{attribute 'reflection'}
FUNCTION_BLOCK PUBLIC FB_DevDoublePWM EXTENDS FB_DevBase // PWM control for 2 outputs that cannot be switchid on simultaniously
VAR_INPUT
	bCmdPWMOn			: BOOL := FALSE ; // PWM controller on 
END_VAR
VAR_OUTPUT
END_VAR
VAR
	bCmdChanelAOn		: BOOL := FALSE ; // command switch chanel A on permanently
	bCmdChanelBOn		: BOOL := FALSE ; // Commandswitch chanel B on permanently 
	bCmdOverrulePWM		: BOOL := FALSE ; // Command to overrule PWM
	bCmdHold			: BOOL := false ; // Command hold PWM on signals (collision avoidance)

	tPeriodLength		: TIME  ; // desired PWM cycle time length [ms] 
	tDutyCycle 			: TIME	; // percentage of power [%]
	tIdleTime			: TIME	; // Time both outputs are idle during PWM
	
	tonOutputA 			: TON ; // Timer on PWM output A
	tonOutputB 			: TON ; // Timer on PWM output B
	tonIdle				: TON ; // Timer On PWM Idle time (both outputs off)

	tofOutputA 			: TOF ; // Timer off PWM output A Off (For overlap prevention)
	tofOutputB 			: TOF ; // Timer off PWM output B Off ( for overlap prevention)

	stParPeriodLength	: Udt_Parameter := (fValue := 2000); // desired PWM cycle time length [ms] Parameter
	stParDutyCycle 		: Udt_Parameter	:= ( fValue := 0); // percentage of power [%] Parameter
	stParSwitchOverTime	: Udt_Parameter	; // Time between switching A off and B on (and vice versa) Parameter
	stMaxTimeOn			: Udt_Parameter := (fValue := 1000);// Maximum time a heater can be on without burning through
	
	qbOutputMain AT %Q* 	: BOOL 	; // physical output to main relais
	qbOutputA	 AT %Q* 	: BOOL 	; // physical output to output A
	qbOutputB	 AT %Q* 	: BOOL 	; // physical output to output B
	
	nPWMStep	: INT ; // PWM stepper

	tonBurnTimeA	: TON ; // burn timer for coil A
	tonBurnTimeB	: TON ; // burn timer for coil B 
END_VAR

// set device type
IF eDevType = E_Devices.Undefined THEN 
	eDevType := E_Devices.DoublePWMController ;
END_IF

// Call base function
SUPER^();


// ===== hold all actions if not initialized ======
IF NOT bInitOk THEN
	RETURN;
END_IF 

// call Functions 
CalcCycleTimes();
IF tDutyCycle > T#0S AND tPeriodLength > T#0S THEN // switch PWM controller up when cycle timer is null
	ExecPWMCycle(); // 
END_IF 

ExecSetOutputs();

METHOD INTERNAL CalcCycleTimes : BOOL // calculate cycle timers
VAR_INPUT
END_VAR
VAR 
END_VAR
// Calculate Cycle timers
tPeriodLength	:= LREAL_TO_TIME( stParPeriodLength.fValue );
tDutyCycle		:= LREAL_TO_TIME(stParPeriodLength.fValue * (stParDutyCycle.fValue / 100));
tIdleTime		:= LREAL_TO_TIME(stParPeriodLength.fValue) - (tDutyCycle * 2) ;

tofOutputA.PT := LREAL_TO_TIME(stParSwitchOverTime.fValue);
tofOutputB.PT := LREAL_TO_TIME(stParSwitchOverTime.fValue);
END_METHOD

METHOD PUBLIC CmdHold : BOOL
VAR_INPUT
END_VAR
bCmdHold := TRUE ;

CmdHold := NOT qbOutputMain ;
END_METHOD

METHOD PUBLIC CmdOutputAOn : BOOL // Turn on chanel A permanently 
VAR_INPUT
END_VAR
bCmdOverrulePWM S= TRUE ;
bCmdChanelAOn S= TRUE ;

CmdOutputAOn := qbOutputA AND qbOutputMain ;
END_METHOD

METHOD PUBLIC CmdOutputBOn : BOOL
VAR_INPUT
END_VAR
bCmdOverrulePWM S= TRUE ;
bCmdChanelBOn S= TRUE ;

CmdOutputBOn := qbOutputB AND qbOutputMain ;
END_METHOD

METHOD PUBLIC CmdSafeStop : BOOL
VAR_INPUT
END_VAR
bCmdOverrulePWM S= TRUE ;
bCmdChanelAOn 		:= FALSE ;
bCmdChanelBOn		:= FALSE ;
qbOutputMain 		:= FALSE ;

bIsSafe := NOT (qbOutputA OR qbOutputB OR qbOutputMain);
END_METHOD

METHOD INTERNAL ExecPWMCycle : BOOL
VAR_INPUT
END_VAR
IF bCmdPWMOn THEN 
	IF bCmdOverrulePWM OR bCmdHold THEN 
		IF bCmdChanelAOn THEN 
			nPWMStep := 1 ;
		ELSE 
			nPWMStep := 0 ;
		END_IF
		bCmdOverrulePWM := FALSE ;
		RETURN;
	END_IF
ELSE 
	RETURN;
END_IF

// PWM stepper 
CASE nPWMStep OF 
	0: // Switch on chanel A
		bCmdChanelAOn := TRUE ;
		IF tonOutputA.Q THEN
			nPWMStep := 1 ;
		END_IF
	1: // Switch on chanel B
		bCmdChanelBOn := TRUE;
		IF tonOutputB.Q THEN
			nPWMStep := 2 ;
		END_IF
	2: // Idle Time 
		IF tonIdle.Q THEN 
			nPWMStep := 0;
		END_IF
	ELSE
		;
END_CASE

// call timers 
tonOutputA	(IN := bCmdChanelAOn, PT := tDutyCycle);
tonOutputB	(IN := bCmdChanelBOn, PT := tDutyCycle);
tonIdle 	(IN := nPWMStep = 2	, PT := tIdleTime);
END_METHOD

METHOD PRIVATE ExecSetOutputs : BOOL
VAR_INPUT
END_VAR

// Set main output
qbOutputMain := (bEnable OR bManual) AND NOT bCmdHold ;

// Set outputs
qbOutputA := bCmdChanelAOn AND NOT tofOutputB.Q AND NOT tonBurnTimeA.Q;
qbOutputB := bCmdChanelBOn AND NOT tofOutputA.Q AND NOT tonBurnTimeB.Q;

// Call timers for overlap prevention
tofOutputA(IN := qbOutputA);
tofOutputB(IN := qbOutputB);

// reset commands
bCmdChanelAOn := FALSE ;
bCmdChanelBOn := FALSE ;

tonBurnTimeA ( IN := bCmdChanelAOn, PT := LREAL_TO_TIME( stMaxTimeOn.fValue));
tonBurnTimeB ( IN := bCmdChanelBOn, PT := LREAL_TO_TIME( stMaxTimeOn.fValue));

IF tonBurnTimeA.Q THEN 
	stFault.Active 			:= TRUE ;
	stFault.Description 	:= 'Heater A burn timeout';
	stFault.FaultType		:= E_FaultTypes.CF;
	qbOutputA 				:= FALSE ;
ELSIF tonBurnTimeB.Q THEN 
	stFault.Active 			:= TRUE ;
	stFault.Description 	:= 'Heater B burn timeout';
	stFault.FaultType		:= E_FaultTypes.CF;
	qbOutputB 				:= FALSE ;
END_IF

bCmdHold := FALSE ;
END_METHOD

METHOD PUBLIC Init : BOOL
VAR_INPUT
	// Message location data
	nId			: UINT ; // Identification number of object
	nParentId	: UDINT ; // Id of higher level If aplicable (0 = no parent)
END_VAR
// ====== Set init to true =====
	bInitOk	:= TRUE ; 

// ====== Calculate device id =====
	bInitOk :=	ExecIdentifyDevice(nId,nParentId, E_ComponentTypes.Heaters) AND bInitOk;

// ======= Reset Error bit ======
	bErrorActive 	:= FALSE;
	bBusy			:= FALSE;
	
// ===== configure parameters =====
	stParPeriodLength.fMinimum 		:= 0 		;
	stParPeriodLength.fMaximum		:= 60000 	;
	stParPeriodLength.nNumber 		:= stIdentity.nLocationId + 1;
	stParPeriodLength.sDiscription  := CONCAT( STR1 := stIdentity.sName, STR2 := ' period length of the cycle');
	stParPeriodLength.sName			:= CONCAT( STR1 := stIdentity.sName, STR2 := 'Period Length');
	stParPeriodLength.sType			:= 'MPar';
	stParPeriodLength.sUnit			:= 'ms';
	stParPeriodLength.fValue		:= 5000;

	stParDutyCycle.fMinimum 		:= 0 		;
	stParDutyCycle.fMaximum			:= 50 		;
	stParDutyCycle.nNumber 			:= stIdentity.nLocationId + 2;
	stParDutyCycle.sDiscription  	:= CONCAT( STR1 := stIdentity.sName, STR2 := ' percentage of period length in which an output is active');
	stParDutyCycle.sName			:= CONCAT( STR1 := stIdentity.sName, STR2 := 'Duty Cyle');
	stParDutyCycle.sType			:= 'MPar';
	stParDutyCycle.sUnit			:= '%';
	stParPeriodLength.fValue		:= 10;

	
	stParSwitchOverTime.fMinimum 	:= 0 		;
	stParSwitchOverTime.fMaximum	:= 500 		;
	stParSwitchOverTime.nNumber 	:= stIdentity.nLocationId + 3;
	stParSwitchOverTime.sDiscription:= CONCAT( STR1 := stIdentity.sName, STR2 := ' idle time between output chanel switchover');
	stParSwitchOverTime.sName		:= CONCAT( STR1 := stIdentity.sName, STR2 := 'Switch Time');
	stParSwitchOverTime.sType		:= 'CPar';
	stParSwitchOverTime.sUnit		:= 'ms';

	stMaxTimeOn.fMinimum 	:= 0 		;
	stMaxTimeOn.fMaximum	:= 5000 	;
	stMaxTimeOn.nNumber 	:= stIdentity.nLocationId + 4;
	stMaxTimeOn.sDiscription:= CONCAT( STR1 := stIdentity.sName, STR2 := ' maximum time a heater can be fully on without burning through');
	stMaxTimeOn.sName		:= CONCAT( STR1 := stIdentity.sName, STR2 := 'Max heating time');
	stMaxTimeOn.sType		:= 'MPar';
	stMaxTimeOn.sUnit		:= 'ms';
	
	
	// add parameters to handler 
	refFbParHandler.CmdAddParameter( refParameter := stParPeriodLength );
	refFbParHandler.CmdAddParameter( refParameter := stParDutyCycle );
	refFbParHandler.CmdAddParameter( refParameter := stParSwitchOverTime );
END_METHOD

END_FUNCTION_BLOCK

(* stored: Version 1.1.0.1, ProductVersion 3.1.4024.11
   POU FB_DevDoublePWM: Id {597d6264-d5f7-07b8-20b6-bf7abd467b88}, SpecialFunc None
   Folder Private: Id {8f1901c9-6ed3-0e55-22ef-5b4692e73382}
   Method CalcCycleTimes: Id {c560b553-2e91-0b3f-2513-3eb8c1b8590a}
   Method CmdHold: Id {2aa262df-5d2b-0f65-1301-f8607be7ccf8}
   Method CmdOutputAOn: Id {285facb1-80c0-01b3-3adb-d410c68724cd}
   Method CmdOutputBOn: Id {ade5c8ae-04d5-0f56-3c6a-987947f25504}
   Method CmdSafeStop: Id {191eddc8-da09-0edf-033c-fd42f3b0ec5d}
   Method ExecPWMCycle: Id {7a1c56a1-834a-0185-2358-6154f346b7a0}
   Method ExecSetOutputs: Id {a756e636-5c44-0f4e-25a7-67cef032dabc}
   Method Init: Id {398f5054-4030-04cb-100b-1777db0e2325} *)
